INTERFACE ITF_BufferB

END_INTERFACE

(* stored: Version 1.1.0.1
   Itf ITF_BufferB: Id {887b6997-c26d-4cf1-bafb-eee559c0e8e6} *)
